{attribute 'tc_no_symbol'}
FUNCTION_BLOCK FB_AutoCal//METTLER电子秤
VAR_INPUT
	xExecute		: BOOL;//指令执行
	xAbort			: BOOL;//指令中断
	xEstop			: BOOL;//急停
	xDeviceRunning	: BOOL;
	xResetRequest	: BOOL;//复位操作
	stDeviceOpe		: ST_AutoCalOpe;
	stparIn				: STAutoCal_ParIn;	 
	stSysPar			: ST_AutoCal_SysPar; 
	xAutoMode    	: BOOL;//0:mannal 1:auto
	xIniting    	: BOOL;//初始化过程中  

END_VAR
VAR_OUTPUT
	xDone			: BOOL;(*完成条件满足*)
	xBusy			: BOOL;(*动作正在执行*)
	xRunning	: BOOL;
	xError			: BOOL;(*错误条件满足*)
	eERRORID		: AutoCal_ERROR;
	xRdyCmd			: BOOL;//指令就绪
	xRdy			: BOOL;//初始化完成
	sHmiError	:STRING;
	stParOut		: STAutoCal_ParOut;
END_VAR

VAR
{attribute 'tc_no_symbol'}
	eState: STATE;//当前状态
{attribute 'tc_no_symbol'}
	xAborted: BOOL;(*指令被打断，一般是处于急停中*)
{attribute 'tc_no_symbol'}
	_CalStep	:INT;//校准流程
{attribute 'tc_no_symbol'}
	_CurrentPumpController	:INT:=1;//当前控制器
{attribute 'tc_no_symbol'}
	_CurrentPumpHead	:INT:=1;//当前泵头
{attribute 'tc_no_symbol'}
	_first :BOOL;
{attribute 'tc_no_symbol'}		
	_xModeChange:BOOL;
{attribute 'tc_no_symbol'}
	_fManual:F_TRIG;
{attribute 'tc_no_symbol'}
	_rManual:R_TRIG;
{attribute 'tc_no_symbol'}	
	i:INT;
{attribute 'tc_no_symbol'}		
	xFirstInvocation:BOOL;
{attribute 'tc_no_symbol'}	
	xAutomodeFlag:BOOL;	
{attribute 'tc_no_symbol'}		
	_diCmdState:INT;
{attribute 'tc_no_symbol'}
	eCmd:AutoCal_CMD;
{attribute 'tc_no_symbol'}
	tOperationTimer:TON;
{attribute 'tc_no_symbol'}
	tSteadyTimer:TON;	
{attribute 'tc_no_symbol'}	
	_xAutoOpe:BOOL;
{attribute 'tc_no_symbol'}	
	_xHMIOpe:BOOL;
{attribute 'tc_no_symbol'}	
	_xDone:BOOL;
{attribute 'tc_no_symbol'}	
	_InjectNum	:INT;//
{attribute 'tc_no_symbol'}
	k	:INT;//
{attribute 'tc_no_symbol'}
	xRuDongPumpError	:BOOL;	
END_VAR

VAR_TEMP
{attribute 'tc_no_symbol'}
	xAgain: BOOL;

END_VAR

VAR

END_VAR


IF NOT _first 
THEN
	_first := TRUE;

ELSE
	xAgain:=0;	
//检测是否允许指令控制(初始状态，没有报警发生)	
	xRdyCmd := eState = STATE.DORMANT AND eERRORID = AutoCal_ERROR.No_ERROR;
	xDone:=_xDone AND xExecute;	
	//检测是否有模式变化
_fManual(CLK:=xAutoMode);
_rManual(CLK:=xAutoMode);
//

IF eState <> STATE.DORMANT//只有在运行的时候，才会检测是否有模式切换发生
THEN
	IF _fManual.Q OR _rManual.Q
	THEN
		_xModeChange := TRUE;
	END_IF
END_IF
	REPEAT
		CASE eState OF
			STATE.DORMANT:
				HandleDormantState(xAgain=> xAgain);
			STATE.EXECUTING:
				HandleExecutingState(xAgain=> xAgain);
			STATE.DONE:
				HandleDoneState(xAgain=> xAgain);
			STATE.INERROR:
				HandleErrorState(xAgain=> xAgain);
			STATE.ABORTING:
				HandleAbortingState(xAgain=> xAgain);
			STATE.ABORTED:
				HandleAbortedState(xAgain=> xAgain);
			STATE.RESETING:
				HandleResettingState(xAgain=> xAgain);
			END_CASE
	UNTIL (xAgain=0)
	END_REPEAT
END_IF


//报错内容输出
CASE eERRORID OF
	AutoCal_ERROR.FLT_AutoMode:
		sHmiError:='FLT_AutoMode';
	AutoCal_ERROR.FLT_CmdTimeOut:
		sHmiError:='FLT_CmdTimeOut';	
	AutoCal_ERROR.FLT_MT_MCK204C:
		sHmiError:='FLT_MT_MCK204C';	
	AutoCal_ERROR.FLT_PARA:
		sHmiError:='FLT_PARA';	
	AutoCal_ERROR.FLT_RudongPump:
		sHmiError:='FLT_RudongPump';	
	AutoCal_ERROR.No_ERROR:
		sHmiError:='No_ERROR';
END_CASE




_xAutoOpe:=stDeviceOpe.x96PumpHeadCal_Auto OR
					stDeviceOpe.xSpecificPumpHeadCal_Auto;
_xHMIOpe:=stDeviceOpe.x96PumpHeadCal_HMI OR
					stDeviceOpe.xContinuesInject_HMI OR
					stDeviceOpe.xInit_Hmi OR
					stDeviceOpe.xSpecificPumpHeadCal_HMI;

{attribute 'tc_no_symbol'}
METHOD PROTECTED AbortAction
VAR_INPUT
END_VAR
VAR_OUTPUT
	xComplete: BOOL;
	eErrorID: AutoCal_ERROR;
END_VAR
(*
* Cleaning
* => abort all running operation
* => if an NBS.ERROR codition is reached, set eErrorID to a Value rather then NBS.ERROR.NO_ERROR 
*)
xComplete:=1;
eErrorID:=AutoCal_ERROR.NO_ERROR;
END_METHOD

ACTION ACT_DensityConversion:
{attribute 'tc_no_symbol'}
//密度计算公式，ρ＝m/V 
IF stParIn.rDensity<>0 THEN
	stParOut.rVolume:=stParOut.rSteadyWeight/stParIn.rDensity;
ELSE
	stParOut.rVolume:=0;
END_IF
END_ACTION

METHOD PROTECTED Cmd_ContinuesInject : BOOL
VAR_INPUT
END_VAR
VAR_OUTPUT
	xComplete: BOOL;
END_VAR
// return the real actual fault number
IF eERRORID <> AutoCal_ERROR.No_ERROR
THEN
  RETURN;  
END_IF
stParOut.iCalStep:=_diCmdState;//流程步输出

CASE _diCmdState OF	
	
		
	0://判断是否到达校准位置
		_diCmdState:=_diCmdState+1;	
			
	1://判断是否结束
	IF _InjectNum<=stparIn.iContinuesInjectNum THEN
		_diCmdState:=_diCmdState+1;
	ELSE
		_diCmdState:=30;//结束加液
	END_IF				
	
	2://等待秤Ready
		IF stsyspar.fbMTMCK204C^.xRdyCmd AND stsyspar.fbRuDongPump[stparIn.iPumpController-1].xRdyCmd THEN
			_diCmdState:=_diCmdState+1;	
		END_IF
	
	3://秤体清零
		stsyspar.fbMTMCK204C^.stDeviceOpe.xShelling_Auto:=TRUE;
		IF stsyspar.fbMTMCK204C^.xDone THEN
			stsyspar.fbMTMCK204C^.xExecute:=FALSE;
			_diCmdState:=_diCmdState+1;
		END_IF

	4://等待稳定时间
		tSteadyTimer(IN:=stsyspar.fbMTMCK204C^.xRdyCmd,PT:=T#1S);
		IF tSteadyTimer.Q THEN
			tSteadyTimer(IN:=FALSE);
			_diCmdState:=_diCmdState+1;
		END_IF	
	
	5://蠕动泵加液
		stsyspar.fbRuDongPump[stparIn.iPumpController-1].stDeviceOpe.xPush_Auto[1]:=TRUE;
		IF stsyspar.fbRuDongPump[stparIn.iPumpController-1].xDone THEN
			stsyspar.fbRuDongPump[stparIn.iPumpController-1].xExecute:=FALSE;
			_diCmdState:=_diCmdState+1;
		END_IF

	6://等待稳定时间
		tSteadyTimer(IN:=stsyspar.fbRuDongPump[stparIn.iPumpController-1].xRdyCmd,PT:=TO_TIME((stparIn.tSteadyTime +stsyspar.fbRuDongPump[stparIn.iPumpController-1].stRunPara.rPushRuntime[1])*1000 ));
		IF tSteadyTimer.Q THEN
			tSteadyTimer(IN:=FALSE);
			_diCmdState:=_diCmdState+1;
		END_IF
	
	7://读取重量
		stsyspar.fbMTMCK204C^.stDeviceOpe.xAcquireWeight_Steady_Auto:=TRUE;
		IF stsyspar.fbMTMCK204C^.xDone THEN
			stsyspar.fbMTMCK204C^.xExecute:=FALSE;
			_diCmdState:=_diCmdState+1;
		END_IF
	
	8://等待稳定时间
		tSteadyTimer(IN:=stsyspar.fbMTMCK204C^.xRdyCmd,PT:=T#1S);
		IF tSteadyTimer.Q THEN
			tSteadyTimer(IN:=FALSE);
			_diCmdState:=_diCmdState+1;
		END_IF		
		
	9://传递重量值
		IF stsyspar.fbMTMCK204C^.stParOut.rCurrentWeight>0 THEN
			stParOut.rContinuesInjectWeight[_InjectNum]:=stsyspar.fbMTMCK204C^.stParOut.rCurrentWeight;
			IF stParOut.rContinuesInjectWeight[_InjectNum]=stsyspar.fbMTMCK204C^.stParOut.rCurrentWeight THEN
				_diCmdState:=_diCmdState+1;
			END_IF
		ELSE
			_diCmdState:=7;
		END_IF		
	
	10://累加
		_InjectNum:=_InjectNum+1;
		_diCmdState:=_diCmdState+1;
	
	11://复位状态
		tSteadyTimer(IN:=TRUE,PT:=T#1S);
		IF tSteadyTimer.Q THEN
			tSteadyTimer(IN:=FALSE);
			_diCmdState:=0;
		END_IF	
		
		
(**************************************************加液结束***************************************************)	
	30://校准完成
		xComplete:=TRUE;
		
	
	
	
	
END_CASE
END_METHOD

METHOD PROTECTED Cmd_Init : BOOL
VAR_INPUT
END_VAR
VAR_OUTPUT
	xComplete: BOOL;
END_VAR
// return the real actual fault number
IF eERRORID <> AutoCal_ERROR.No_ERROR
THEN
  RETURN;  
END_IF
stParOut.iCalStep:=_diCmdState;//流程步输出
CASE _diCmdState OF	
		
	0://
		_CurrentPumpController:=1;//从1#泵开始
		_diCmdState:=10;
(**************蠕动泵停止**************)			
	10://判断N#泵控制器参数
		_CurrentPumpController:=1;//从1#开始
		_diCmdState:=_diCmdState+1;
		
	11://判断是否结束
		IF	_CurrentPumpController>gc_uiRudongPump THEN
			_diCmdState:=20;
		ELSE
			IF stSysPar.fbRuDongPump[_CurrentPumpController-1].xRdyCmd THEN
				_diCmdState:=_diCmdState+1;
			END_IF
		END_IF
		
	12://停止N#泵控制器	
		stSysPar.fbRuDongPump[_CurrentPumpController-1].stDeviceOpe.xStop_Auto:=TRUE;
		IF stSysPar.fbRuDongPump[_CurrentPumpController-1].xDone THEN
			stSysPar.fbRuDongPump[_CurrentPumpController-1].xExecute:=FALSE;
			_diCmdState:=_diCmdState+1;
		END_IF		
	
	13://累加1
		_CurrentPumpController:=_CurrentPumpController+1;
		_diCmdState:=_diCmdState+1;
		
	14://回去循环执行
		_diCmdState:=11;

(**************************************************秤清零***************************************************)	
	20://判断秤体状态
		IF stSysPar.fbMTMCK204C^.xRdyCmd THEN
			_diCmdState:=22;
		ELSE
			IF stSysPar.fbMTMCK204C^.stParOut.xContinuesRead THEN
				_diCmdState:=_diCmdState+1;
			END_IF
		END_IF
	
	21://停止连续读取
			stSysPar.fbMTMCK204C^.stDeviceOpe.xAcquireWeight_Stop_Auto:=TRUE;
			IF stSysPar.fbMTMCK204C^.xRdyCmd THEN
				_diCmdState:=_diCmdState+1;
			END_IF			

	22://秤重启
			stSysPar.fbMTMCK204C^.stDeviceOpe.xRestart_Auto:=TRUE;
			IF stSysPar.fbMTMCK204C^.xDone THEN
				stSysPar.fbMTMCK204C^.xExecute:=FALSE;
				_diCmdState:=30;
			END_IF			
	

(*************************************************初始化结束***************************************************)
	30://校准完成
		xComplete:=TRUE;
		

	
END_CASE
END_METHOD

METHOD PROTECTED Cmd_SpecificPumpHeadCal : BOOL
VAR_INPUT
END_VAR
VAR_OUTPUT
	xComplete: BOOL;
END_VAR
// return the real actual fault number
IF eERRORID <> AutoCal_ERROR.No_ERROR
THEN
  RETURN;  
END_IF
stParOut.iCalStep:=_diCmdState;//流程步输出

CASE _diCmdState OF	
	
		
	0://判断是否到达校准位置
		_diCmdState:=_diCmdState+1;	
		
	1://等待校准就绪
		IF stsyspar.fbMTMCK204C^.xRdyCmd AND stsyspar.fbRuDongPump[stparIn.iPumpController-1].xRdyCmd THEN
			_diCmdState:=_diCmdState+1;	
		END_IF		
		
(**************************************************校准***************************************************)		
	2://秤体清零	
		stSysPar.fbMTMCK204C^.stDeviceOpe.xClearZero_Auto:=TRUE;
		IF stSysPar.fbMTMCK204C^.xDone THEN
			stSysPar.fbMTMCK204C^.xExecute:=FALSE;
			_diCmdState:=_diCmdState+1;	
		END_IF
		
	3://等待稳定时间
		tSteadyTimer(IN:=TRUE,PT:=T#1S);
		IF tSteadyTimer.Q THEN
			tSteadyTimer(IN:=FALSE);
			_diCmdState:=_diCmdState+1;
		END_IF		
		
	4://校准启动	
		stSysPar.fbRuDongPump[_CurrentPumpController-1].stDeviceOpe.xPumpCal_Auto:=TRUE;
		IF stSysPar.fbRuDongPump[_CurrentPumpController-1].xDone THEN
			stSysPar.fbMTMCK204C^.xExecute:=FALSE;
			_diCmdState:=_diCmdState+1;
		END_IF
		
	5://等待稳定时间
		tSteadyTimer(IN:=TRUE,PT:=TO_TIME((stparIn.tSteadyTime+1)*1000));
		IF tSteadyTimer.Q THEN
			_diCmdState:=_diCmdState+1;
		END_IF

	6://获取称重结果
			stSysPar.fbMTMCK204C^.stDeviceOpe.xAcquireWeight_Steady_Auto:=TRUE;
			IF stSysPar.fbMTMCK204C^.xDone THEN
				stSysPar.fbMTMCK204C^.xExecute:=FALSE;
				_diCmdState:=_diCmdState+1;	
			END_IF	
	
	7://等待稳定时间
		tSteadyTimer(IN:=TRUE,PT:=T#1S);
		IF tSteadyTimer.Q THEN
			tSteadyTimer(IN:=FALSE);
			_diCmdState:=_diCmdState+1;
		END_IF			

	8://获取称重结果
		IF stSysPar.fbMTMCK204C^.stParOut.rCurrentWeight>0 THEN
			stParOut.rSteadyWeight:=stSysPar.fbMTMCK204C^.stParOut.rCurrentWeight;
			IF stParOut.rSteadyWeight=stSysPar.fbMTMCK204C^.stParOut.rCurrentWeight THEN
				_diCmdState:=_diCmdState+1;
			END_IF
		ELSE
			_diCmdState:=6;//未获取到重量重新读
		END_IF
		
	9://给校准参数赋值
		stSysPar.fbRuDongPump^.stRunPara.rModuleRealFluVolume:=stParOut.rVolume;
		stSysPar.fbRuDongPump^.stDeviceOpe.xCalParWrite_Auto:=TRUE;
		IF stSysPar.fbRuDongPump^.xDone THEN
			_diCmdState:=30;
		END_IF
	

(**************************************************校准结束***************************************************)	
	30://校准完成
		xComplete:=TRUE;
		
	
	
	
	
END_CASE
END_METHOD

{attribute 'tc_no_symbol'}
METHOD PROTECTED CyclicAction
VAR_INPUT
END_VAR
VAR_OUTPUT
	xComplete: BOOL;
END_VAR
VAR	
END_VAR
IF xAbort=0 THEN
	IF xFirstInvocation THEN//执行初始化
	(*
	* Staring
	* for then first (!) invocaion,
	* sample then input variables
	*)
		xFirstInvocation:=0;
	END_IF    
	REPEAT 	
//判断是否有参数错误		
		IF stSysPar.fbMTMCK204C=0 OR
				stSysPar.fbRuDongPump=0 OR
				stSysPar.iRuDongPumpHeadNum>32
		THEN
			eERRORID:=AutoCal_ERROR.FLT_PARA;//参数配置错误
		ELSE
			xRuDongPumpError:=FALSE;
			FOR k:=1 TO gc_uiRudongPump DO
				IF stSysPar.fbRuDongPump[k].xError THEN
					xRuDongPumpError:=TRUE;
					EXIT;
				END_IF
			END_FOR			

			//IF stSysPar.fbMTMCK204C^.xError THEN
			//	eERRORID:=AutoCal_ERROR.FLT_MT_MCK204C;//秤出错
			//ELSE
			//	IF xRuDongPumpError THEN
			//		eERRORID:=AutoCal_ERROR.FLT_RudongPump;//蠕动泵出错
			//	END_IF						
			//END_IF
		END_IF

			//如果不在自动模式则报错
			IF _xAutoOpe OR _xHMIOpe THEN
					xRunning:=TRUE;
			END_IF

			CASE eCmd OF//判断指令类型
				AutoCal_CMD.Cmd_SpecificPumpHeadCal://单个泵头校准
					Cmd_SpecificPumpHeadCal(xComplete=> xComplete);	
				AutoCal_CMD.Cmd_Init://初始化
					Cmd_Init(xComplete=> xComplete);	
				AutoCal_CMD.Cmd_ContinuesInject://连续加液测试
					Cmd_ContinuesInject(xComplete=> xComplete);
					;				
				
			ELSE
				;	
			END_CASE
	   
		UNTIL (TRUE)//处于一直刷新阶段
	END_REPEAT
END_IF

IF NOT xExecute OR xComplete OR eErrorID<>AutoCal_ERROR.No_ERROR THEN    
    (*
    * Cleaning
    * => free as much allocated resources as possible
    *)    
    tOperationTimer(IN:=0);
END_IF
END_METHOD

{attribute 'tc_no_symbol'}
METHOD PRIVATE FINAL HandleAbortedSTATE
VAR_INPUT
END_VAR
VAR_OUTPUT
	xAgain: BOOL;
END_VAR
VAR
	xComplete: BOOL;
END_VAR
IF xAborted AND xResetRequest THEN
    eState:=STATE.RESETING;
    xAgain:=1;
ELSE
    xBusy:=0;
    xAborted:=1;
    //xResetRequest:=(xExecute=0);
    xAgain:=0;(* !!! *)
END_IF
END_METHOD

{attribute 'tc_no_symbol'}
METHOD PRIVATE FINAL HandleAbortingSTATE
VAR_INPUT
END_VAR
VAR_OUTPUT
	xAgain: BOOL;
END_VAR
VAR
{attribute 'tc_no_symbol'}	
	xComplete: BOOL;
END_VAR
AbortAction(xComplete=> xComplete, eErrorID=> eErrorID);

IF eErrorID<>AutoCal_ERROR.NO_ERROR THEN
    eState:=STATE.INERROR;
    xAgain:=1;
ELSIF xComplete THEN
    eState:=STATE.ABORTED;
    xAgain:=1;
END_IF
END_METHOD

{attribute 'tc_no_symbol'}
METHOD PRIVATE FINAL HandleDoneSTATE
VAR_INPUT
END_VAR
VAR_OUTPUT
	xAgain: BOOL;
END_VAR
//在运行过程中要是切换模式，再运行完成之后，检测到模式的切换，就需要回到初始位置，进行下一次执行准备
IF _xDone AND ((xExecute=0) OR ( _xModeChange AND NOT _xAutoOpe)  OR ( NOT xAutoMode AND NOT xDeviceRunning AND ( NOT _xAutoOpe OR _xHMIOpe))) THEN
	eState:=STATE.RESETING;
	xAgain:=1;
ELSE
	xBusy:=0;
	_xDone:=1;
	//xResetRequest:=(xExecute=0);
	xAgain:=0;(* !!! *)
END_IF
END_METHOD

{attribute 'tc_no_symbol'}
METHOD PRIVATE FINAL HandleDormantSTATE
VAR_INPUT
END_VAR
VAR_OUTPUT
	xAgain: BOOL;
END_VAR
IF xExecute THEN
    xBusy:=1;
    eState:=STATE.EXECUTING;
    xAgain:=1;
END_IF

IF xResetRequest//清空报警
THEN
	eERRORID := AutoCal_ERROR.No_ERROR;
END_IF
IF  xAutoMode OR xDeviceRunning THEN
	xAutomodeFlag:=TRUE;
ELSE
	xAutomodeFlag:=FALSE;
END_IF
(********************************等待手动操作******************************)


IF eErrorID = AutoCal_ERROR.NO_ERROR AND xEStop
THEN
	
//校准指定泵头
	IF (stDeviceOpe.xSpecificPumpHeadCal_HMI OR stDeviceOpe.xSpecificPumpHeadCal_Auto)THEN//
		_CurrentPumpController:=stparIn.iPumpController;
		_CurrentPumpHead:=stparIn.iPumpHead;
		eCmd := AutoCal_CMD.Cmd_SpecificPumpHeadCal;
		xExecute := TRUE;
	END_IF
//初始化校准程序
	IF stDeviceOpe.xInit_Hmi THEN//
		eCmd := AutoCal_CMD.Cmd_Init;
		xExecute := TRUE;
	END_IF	
	
//连续加液测试
	IF stDeviceOpe.xContinuesInject_HMI THEN//
		FOR i:=1 TO 30 DO
			stParOut.rContinuesInjectWeight[i]:=0;
		END_FOR
		_InjectNum:=1;
		eCmd := AutoCal_CMD.Cmd_ContinuesInject;
		xExecute := TRUE;
	END_IF	
	
END_IF
END_METHOD

{attribute 'tc_no_symbol'}
METHOD PRIVATE FINAL  HandleErrorSTATE
VAR_INPUT
END_VAR
VAR_OUTPUT
	xAgain: BOOL;
END_VAR
IF xError AND  (xResetRequest OR NOT xExecute) THEN
    eState:=STATE.RESETING;
    xAgain:=1;
ELSE
    xBusy:=0;
    xError:=1;    
    xAgain:=0;(* !!! *)
END_IF
END_METHOD

{attribute 'tc_no_symbol'}
METHOD PRIVATE FINAL HandleExecutingSTATE
VAR_INPUT
END_VAR
VAR_OUTPUT
	xAgain: BOOL;
END_VAR
VAR
{attribute 'tc_no_symbol'}	
	xComplete: BOOL;
END_VAR

IF xAbort=0 THEN   
    CyclicAction(xComplete=> xComplete);
END_IF

IF eErrorID<>AutoCal_ERROR.NO_ERROR THEN
    eState:=STATE.INERROR;
    xAgain:=1;
ELSIF xAbort THEN
    eState:=STATE.ABORTING;
    xAgain:=1;
ELSIF xComplete THEN
    eState:=STATE.DONE;
    xAgain:=1;
END_IF
END_METHOD

{attribute 'tc_no_symbol'}
METHOD PRIVATE FINAL HandleResettingSTATE
VAR_INPUT
END_VAR
VAR_OUTPUT
	xAgain: BOOL;
END_VAR
VAR
{attribute 'tc_no_symbol'}	
	xComplete: BOOL;
END_VAR
ResetAction(xComplete=> xComplete);

IF xComplete THEN
		xExecute:=0;//清除输入指令 
    xBusy:=0;
    xDone:=0;
    xError:=0;

    eErrorID:=AutoCal_ERROR.NO_ERROR;
    eState:=STATE.DORMANT;
    xFirstInvocation:=1;
    xAgain:=0;(* !!! *)
END_IF
END_METHOD

{attribute 'tc_no_symbol'}
METHOD PROTECTED ResetAction
VAR_INPUT
END_VAR
VAR_OUTPUT
	xComplete: BOOL;
END_VAR
(*
* Cleaning
* => free all allocated resources
* => reinitialize instance variables
*)
tOperationTimer(IN:=0);
_diCmdState:=0;
_CurrentPumpController:=1;
stDeviceOpe.x96PumpHeadCal_Auto:=
stDeviceOpe.x96PumpHeadCal_HMI:=
stDeviceOpe.xInit_Auto:=
stDeviceOpe.xInit_Hmi:=
stDeviceOpe.xSpecificPumpHeadCal_Auto:=
stDeviceOpe.xContinuesInject_HMI:=
stDeviceOpe.xSpecificPumpHeadCal_HMI:=FALSE;
xRunning:=FALSE; 
xComplete:=1;	

stsyspar.fbRuDongPump[stparIn.iPumpController-1].xExecute:=FALSE;
stsyspar.fbRuDongPump[stparIn.iPumpController-1].stDeviceOpe.xPush_Auto[1]:=TRUE;
stsyspar.fbMTMCK204C^.xExecute:=FALSE;
END_METHOD

END_FUNCTION_BLOCK

(* stored: Version 1.1.0.1, ProductVersion 3.1.4024.9
   POU FB_AutoCal: Id {666d666e-5622-456d-b634-396736292374}, SpecialFunc None
   Folder Control: Id {89e1fc37-6f6a-4b35-a9e7-cec8fe2e71f9}
   Method AbortAction: Id {40c5fd6f-87a9-403a-aca3-e8645c812a00}
   Action ACT_DensityConversion: Id {9656d47a-dbee-49fe-8433-c711d80dd636}
   Method Cmd_ContinuesInject: Id {3e5b722f-fa7b-4887-9f26-cfa9b867f01d}
   Method Cmd_Init: Id {50f3d719-e078-4a6e-b8f9-f6b59207e421}
   Method Cmd_SpecificPumpHeadCal: Id {1cec9c0a-cf09-4f24-bf88-6065c78435b3}
   Method CyclicAction: Id {0fea1345-6f6c-4620-b1bd-e9c33dd9c2e2}
   Method HandleAbortedState: Id {c4be324d-cc71-4443-a6ae-151a688040e9}
   Method HandleAbortingState: Id {02931520-ed5d-41c4-a893-eb29ec4ccedf}
   Method HandleDoneState: Id {90d4ccf9-393c-4fbc-92e5-c92e86958d5b}
   Method HandleDormantState: Id {b077e08a-44a2-46c3-8e9c-df3fd9cf939c}
   Method HandleErrorState: Id {2834be5f-0b02-4f72-a9d0-a241c99e8854}
   Method HandleExecutingState: Id {aba2cef6-09f0-45da-904a-a99c7496a79c}
   Method HandleResettingState: Id {8d7e1e10-f174-46af-b024-96956c089b72}
   Method ResetAction: Id {6acb7093-0bcb-495d-8c5e-582e0a23a161} *)
